INTERFACE I_PackML_CompleteCommands

METHOD PUBLIC Abort
VAR_INPUT
END_VAR
END_METHOD

METHOD PUBLIC Reset
VAR_INPUT
END_VAR
END_METHOD

METHOD PUBLIC Stop
VAR_INPUT
END_VAR
END_METHOD

END_INTERFACE

(* stored: Version 1.1.0.1, ProductVersion 3.1.4024.12
   Itf I_PackML_CompleteCommands: Id {ec0323ba-8561-0e01-188f-98bb79bd5ab9}
   Method Abort: Id {932f44a8-9748-0e44-222a-c2f7449efb7f}
   Method Reset: Id {0a3bd21e-210b-0b21-2287-f384442eb68d}
   Method Stop: Id {2ff6b9d8-7ece-0e6b-11c5-17f65b58aa16} *)
